{attribute 'no_explicit_call' := 'Base is a class, do not call this POU directly, use a method'}
{attribute 'hide_all_locals'}
{attribute 'reflection'}
FUNCTION_BLOCK ABSTRACT Base
VAR
    {attribute 'instance-path'}
    {attribute 'noinit'}
    _path   : T_MAXSTRING;

	// Locals 
   _name   : T_MAXSTRING;
    _logger : I_Logger;
END_VAR

METHOD FB_Init : BOOL
VAR_INPUT
    bInitRetains : BOOL;
    bInCopyCode  : BOOL;
    name         : STRING;
    logger       : I_Logger;
END_VAR
_name   := name;
_logger := logger;
END_METHOD

PROPERTY name : string
GET
name := _name;
END_GET
END_PROPERTY

PROPERTY path : string
GET
path := _path;
END_GET
END_PROPERTY

METHOD trace
VAR_INPUT
    message : T_MAXSTRING;
END_VAR
IF _logger <> 0 THEN
    _logger.trace(message);
ELSE
    ADSLOGSTR(msgCtrlMask := ADSLOG_MSGTYPE_HINT, msgFmtStr := message, strArg := '');
END_IF
END_METHOD

END_FUNCTION_BLOCK

(* stored: Version 1.1.0.1, ProductVersion 3.1.4026.18
   POU Base: Id {691e5c5d-4b10-4eef-86d7-b1ce8df84e2e}, SpecialFunc None
   Method FB_Init: Id {30c63446-bc96-435b-a4f6-0ed3aa33960d}
   Property name: Id {94530714-4f62-43b0-bd5e-6a5ea5273e6e}
   Get Get: Id {d705c8ca-e1b7-4ceb-822c-3f6e442858af}
   Property path: Id {eaa4fbd5-a93a-4421-9eb7-72d1cf6e92c7}
   Get Get: Id {866da755-f670-4e64-a217-cb05c8cd0f62}
   Method trace: Id {c35e6399-ec56-40cf-a279-c2712ea742df} *)
